SUBAPPLICATION Uebung_034_AD (* Analog-Eingang auf PWM Ausgang (Adapter Version) *)
  (* Standard: 61499-2; Description: Copyright (c) 2023 Meisterschulen am Ostbahnhof This program and the accompanying materials are made available under the terms of the Eclipse Public License 2.0 which is available at https://www.eclipse.org/legal/epl-2.0/ SPDX-License-Identifier: EPL-2.0 *)
  (* Version 1.0, 2026-04-20, Franz Höpfinger, Meisterschulen am Ostbahnhof, initial API and implementation (Adapter Version of Uebung_034) *)
  PACKAGE Uebungen;
  IMPORT logiBUS::io::AI::logiBUS_AI;
  IMPORT logiBUS::io::DQ::logiBUS_DO::Output_Q4;
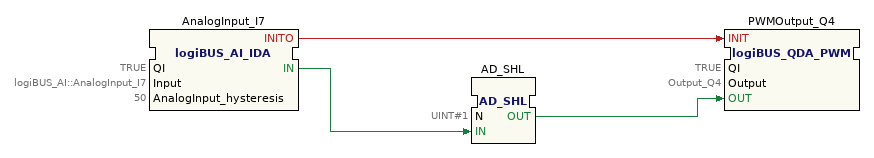
  FBS
    AnalogInput_I7 : logiBUS::io::AI::logiBUS_AI_IDA(QI := TRUE, Input := logiBUS_AI::AnalogInput_I7, AnalogInput_hysteresis := 50);
    PWMOutput_Q4 : logiBUS::io::DQ::logiBUS_QDA_PWM(QI := TRUE, Output := Output_Q4);
    AD_SHL : adapter::iec61131::bitwise::AD_SHL(N := UINT#1);
  END_FBS
  EVENT_CONNECTIONS
    AnalogInput_I7.INITO TO PWMOutput_Q4.INIT;
  END_CONNECTIONS
  ADAPTER_CONNECTIONS
    AnalogInput_I7.IN TO AD_SHL.IN;
    AD_SHL.OUT TO PWMOutput_Q4.OUT;
  END_CONNECTIONS
END_SUBAPPLICATION
